PROGRAM MAIN
VAR
END_VAR

END_PROGRAM

(* stored: Version 1.1.0.1
   POU MAIN: Id {1c723f5a-004e-42fa-96c6-f6989c2b08f3} *)
